FUNCTION_BLOCK FB_GantryDiffVirtualLimitSwitch_Test EXTENDS TcUnit.FB_TestSuite
VAR
    Expected: BOOL;
    Actual: BOOL;
END_VAR

TEST('FB_GantryDiffVirtualLimitSwitch_Test Dummy Test');
AssertEquals(Expected := Expected,
             Actual := Actual,
             Message := 'Error Message');
TEST_FINISHED();

END_FUNCTION_BLOCK

(* stored: Version 1.1.0.1, ProductVersion 3.1.4022.18
   POU FB_GantryDiffVirtualLimitSwitch_Test: Id {a2f81bb8-5c3e-43ea-a1e0-d8fc1eb97af5}, SpecialFunc None *)
